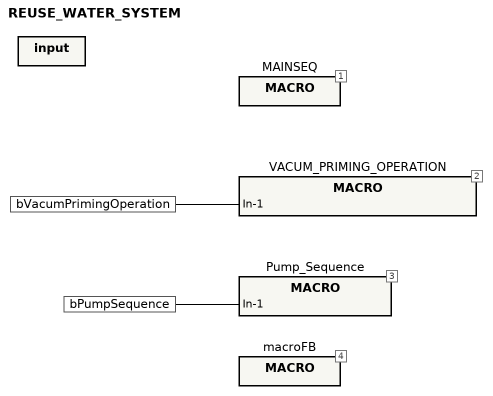
[picture p24: REUSE_WATER_SYSTEM (CFC)]
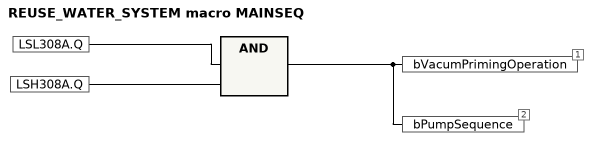
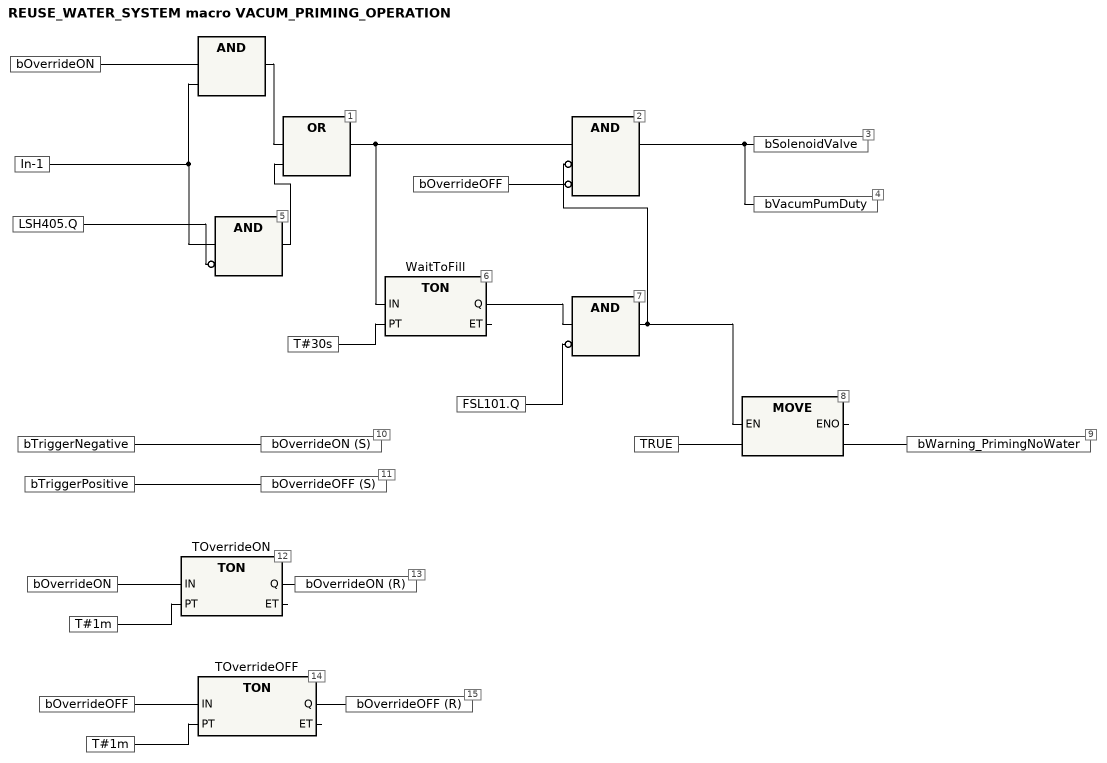
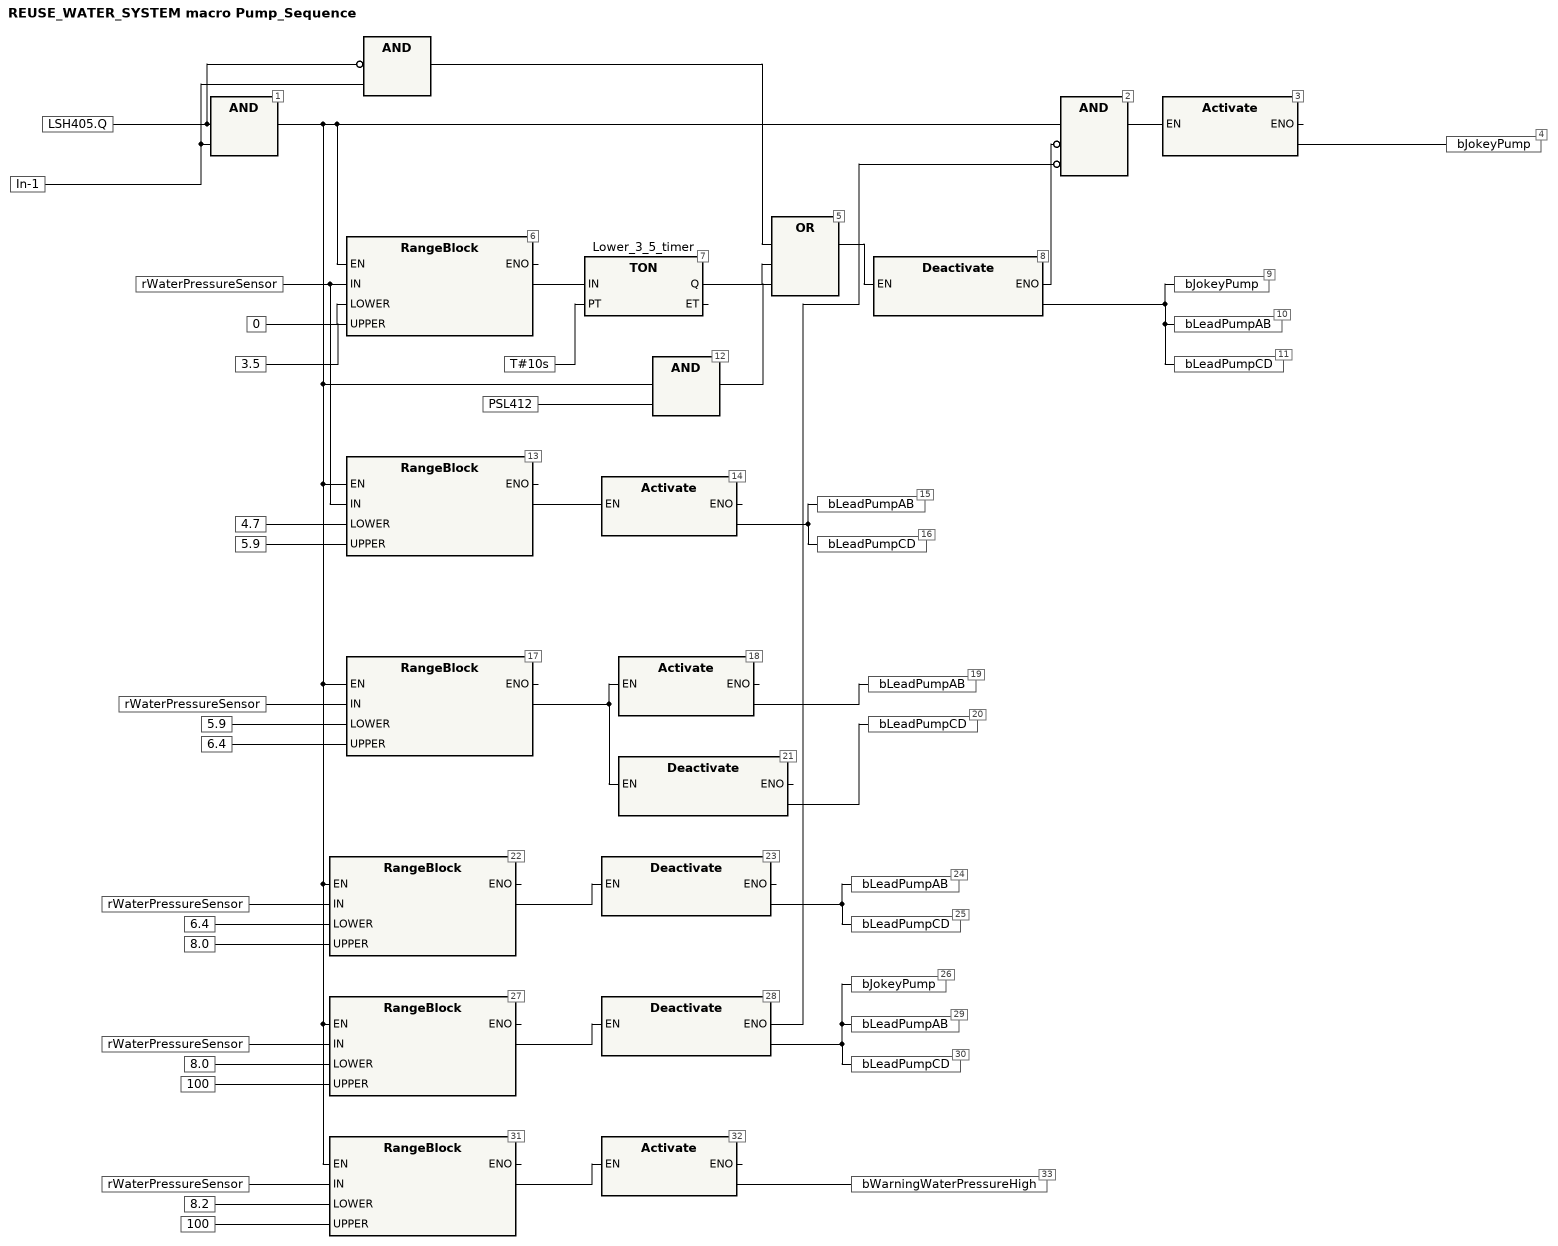
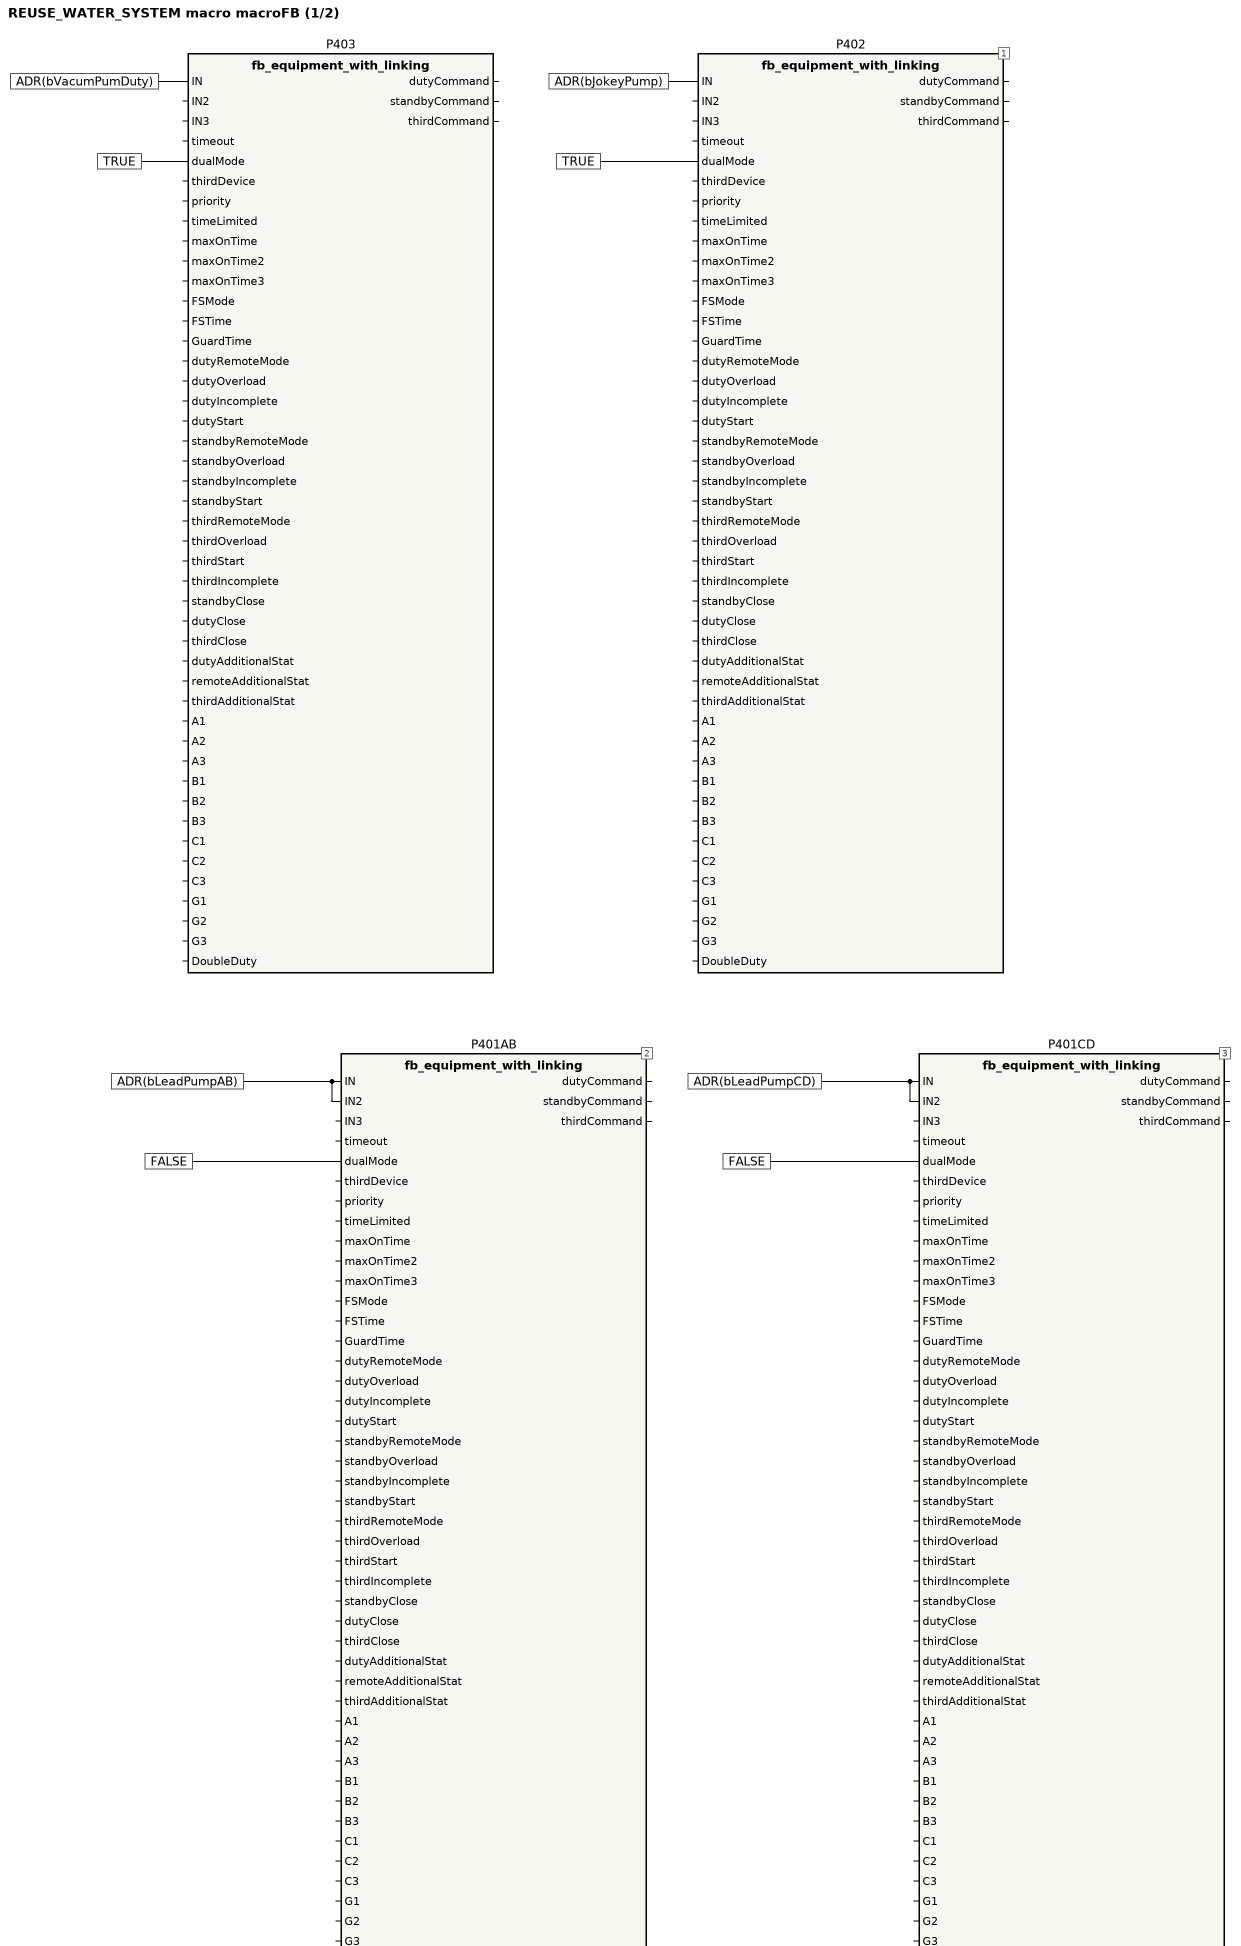
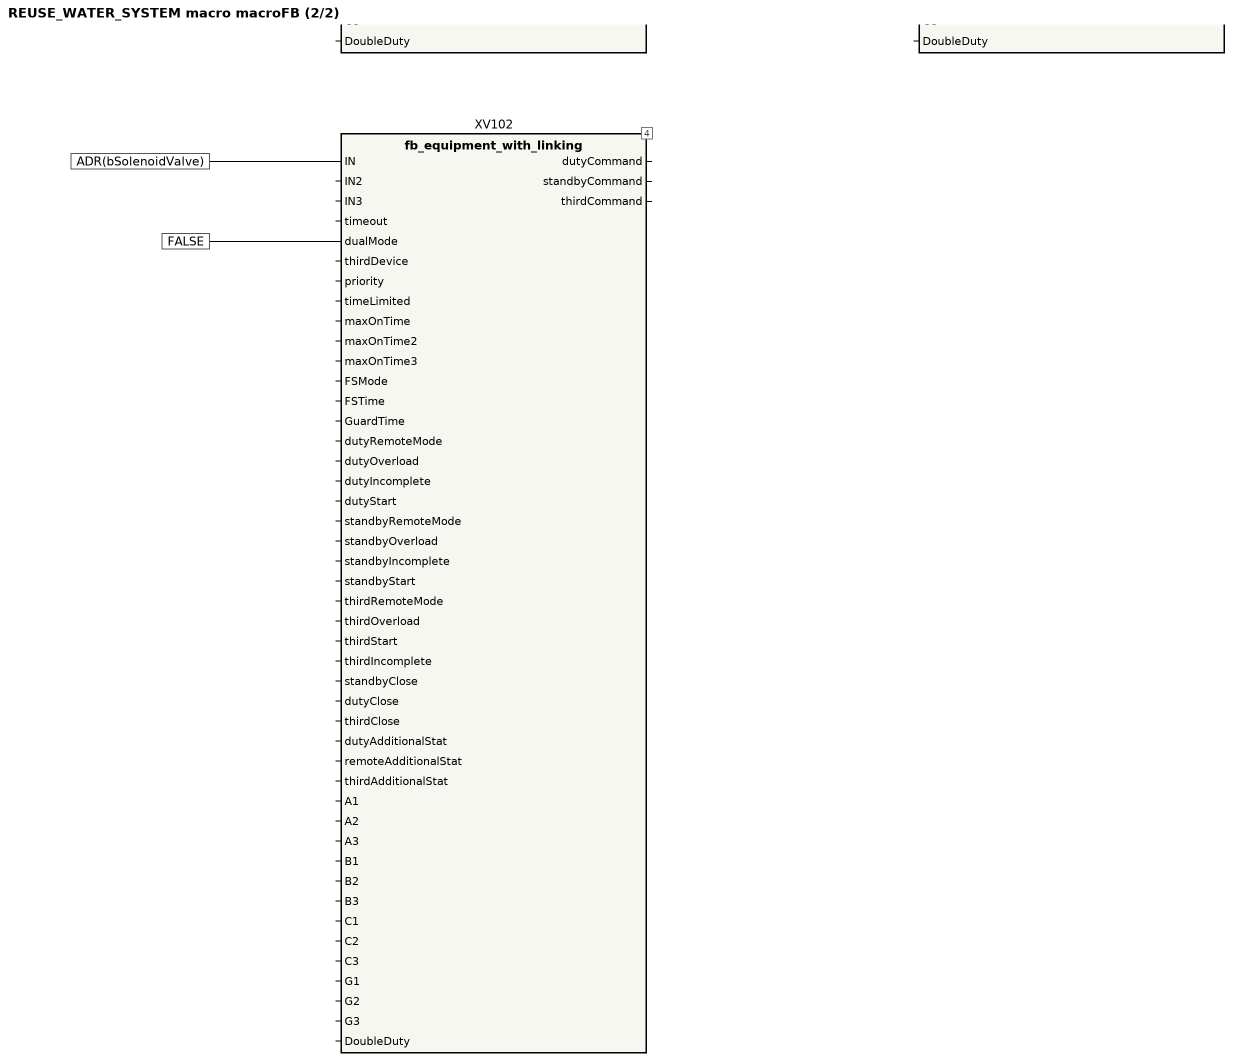
_CFC_ (* Continuous Function Chart, elements in execution order *)
#0 input()
#1 MACRO MAINSEQ()
	#2 AND(LSL308A.Q, LSH308A.Q)
	#3 bVacumPrimingOperation <= #2
	#4 bPumpSequence <= #2
END_MACRO
#5 MACRO VACUM_PRIMING_OPERATION(pin 1 "In-1": bVacumPrimingOperation)
	#6 AND(bOverrideON, pin 1)
	#7 OR(#6, #11)
	#8 AND(#7, NOT #13, NOT bOverrideOFF)
	#9 bSolenoidValve <= #8
	#10 bVacumPumDuty <= #8
	#11 AND(pin 1, NOT LSH405.Q)
	#12 WaitToFill:TON(IN: #7, PT: T#30s)
	#13 AND(#12.Q, NOT FSL101.Q)
	#14 MOVE(EN: #13, TRUE)
	#15 bWarning_PrimingNoWater <= #14
	#16 S bOverrideON <= bTriggerNegative
	#17 S bOverrideOFF <= bTriggerPositive
	#18 TOverrideON:TON(IN: bOverrideON, PT: T#1m)
	#19 R bOverrideON <= #18.Q
	#20 TOverrideOFF:TON(IN: bOverrideOFF, PT: T#1m)
	#21 R bOverrideOFF <= #20.Q
END_MACRO
#22 MACRO Pump_Sequence(pin 1 "In-1": bPumpSequence)
	#23 AND(NOT LSH405.Q, pin 1)
	#24 AND(LSH405.Q, pin 1)
	#25 AND(#24, NOT #31.ENO, NOT #51.ENO)
	#26 Activate(EN: #25)
	#27 bJokeyPump <= #26
	#28 OR(#23, #30.Q, #35)
	#29 RangeBlock(EN: #24, IN: rWaterPressureSensor, LOWER: 0, UPPER: 3.5)
	#30 Lower_3_5_timer:TON(IN: #29, PT: T#10s)
	#31 Deactivate(EN: #28)
	#32 bJokeyPump <= #31
	#33 bLeadPumpAB <= #31
	#34 bLeadPumpCD <= #31
	#35 AND(#24, PSL412)
	#36 RangeBlock(EN: #24, IN: rWaterPressureSensor, LOWER: 4.7, UPPER: 5.9)
	#37 Activate(EN: #36)
	#38 bLeadPumpAB <= #37
	#39 bLeadPumpCD <= #37
	#40 RangeBlock(EN: #24, IN: rWaterPressureSensor, LOWER: 5.9, UPPER: 6.4)
	#41 Activate(EN: #40)
	#42 bLeadPumpAB <= #41
	#43 bLeadPumpCD <= #44
	#44 Deactivate(EN: #40)
	#45 RangeBlock(EN: #24, IN: rWaterPressureSensor, LOWER: 6.4, UPPER: 8.0)
	#46 Deactivate(EN: #45)
	#47 bLeadPumpAB <= #46
	#48 bLeadPumpCD <= #46
	#49 bJokeyPump <= #51
	#50 RangeBlock(EN: #24, IN: rWaterPressureSensor, LOWER: 8.0, UPPER: 100)
	#51 Deactivate(EN: #50)
	#52 bLeadPumpAB <= #51
	#53 bLeadPumpCD <= #51
	#54 RangeBlock(EN: #24, IN: rWaterPressureSensor, LOWER: 8.2, UPPER: 100)
	#55 Activate(EN: #54)
	#56 bWarningWaterPressureHigh <= #55
END_MACRO
#57 MACRO macroFB()
	#58 P403:fb_equipment_with_linking(IN: ADR(bVacumPumDuty), IN2: -, IN3: -, timeout: -, dualMode: TRUE, thirdDevice: -, priority: -, timeLimited: -, maxOnTime: -, maxOnTime2: -, maxOnTime3: -, FSMode: -, FSTime: -, GuardTime: -, dutyRemoteMode: -, dutyOverload: -, dutyIncomplete: -, dutyStart: -, standbyRemoteMode: -, standbyOverload: -, standbyIncomplete: -, standbyStart: -, thirdRemoteMode: -, thirdOverload: -, thirdStart: -, thirdIncomplete: -, standbyClose: -, dutyClose: -, thirdClose: -, dutyAdditionalStat: -, remoteAdditionalStat: -, thirdAdditionalStat: -, A1: -, A2: -, A3: -, B1: -, B2: -, B3: -, C1: -, C2: -, C3: -, G1: -, G2: -, G3: -, DoubleDuty: -)
	#59 P402:fb_equipment_with_linking(IN: ADR(bJokeyPump), IN2: -, IN3: -, timeout: -, dualMode: TRUE, thirdDevice: -, priority: -, timeLimited: -, maxOnTime: -, maxOnTime2: -, maxOnTime3: -, FSMode: -, FSTime: -, GuardTime: -, dutyRemoteMode: -, dutyOverload: -, dutyIncomplete: -, dutyStart: -, standbyRemoteMode: -, standbyOverload: -, standbyIncomplete: -, standbyStart: -, thirdRemoteMode: -, thirdOverload: -, thirdStart: -, thirdIncomplete: -, standbyClose: -, dutyClose: -, thirdClose: -, dutyAdditionalStat: -, remoteAdditionalStat: -, thirdAdditionalStat: -, A1: -, A2: -, A3: -, B1: -, B2: -, B3: -, C1: -, C2: -, C3: -, G1: -, G2: -, G3: -, DoubleDuty: -)
	#60 P401AB:fb_equipment_with_linking(IN: ADR(bLeadPumpAB), IN2: ADR(bLeadPumpAB), IN3: -, timeout: -, dualMode: FALSE, thirdDevice: -, priority: -, timeLimited: -, maxOnTime: -, maxOnTime2: -, maxOnTime3: -, FSMode: -, FSTime: -, GuardTime: -, dutyRemoteMode: -, dutyOverload: -, dutyIncomplete: -, dutyStart: -, standbyRemoteMode: -, standbyOverload: -, standbyIncomplete: -, standbyStart: -, thirdRemoteMode: -, thirdOverload: -, thirdStart: -, thirdIncomplete: -, standbyClose: -, dutyClose: -, thirdClose: -, dutyAdditionalStat: -, remoteAdditionalStat: -, thirdAdditionalStat: -, A1: -, A2: -, A3: -, B1: -, B2: -, B3: -, C1: -, C2: -, C3: -, G1: -, G2: -, G3: -, DoubleDuty: -)
	#61 P401CD:fb_equipment_with_linking(IN: ADR(bLeadPumpCD), IN2: ADR(bLeadPumpCD), IN3: -, timeout: -, dualMode: FALSE, thirdDevice: -, priority: -, timeLimited: -, maxOnTime: -, maxOnTime2: -, maxOnTime3: -, FSMode: -, FSTime: -, GuardTime: -, dutyRemoteMode: -, dutyOverload: -, dutyIncomplete: -, dutyStart: -, standbyRemoteMode: -, standbyOverload: -, standbyIncomplete: -, standbyStart: -, thirdRemoteMode: -, thirdOverload: -, thirdStart: -, thirdIncomplete: -, standbyClose: -, dutyClose: -, thirdClose: -, dutyAdditionalStat: -, remoteAdditionalStat: -, thirdAdditionalStat: -, A1: -, A2: -, A3: -, B1: -, B2: -, B3: -, C1: -, C2: -, C3: -, G1: -, G2: -, G3: -, DoubleDuty: -)
	#62 XV102:fb_equipment_with_linking(IN: ADR(bSolenoidValve), IN2: -, IN3: -, timeout: -, dualMode: FALSE, thirdDevice: -, priority: -, timeLimited: -, maxOnTime: -, maxOnTime2: -, maxOnTime3: -, FSMode: -, FSTime: -, GuardTime: -, dutyRemoteMode: -, dutyOverload: -, dutyIncomplete: -, dutyStart: -, standbyRemoteMode: -, standbyOverload: -, standbyIncomplete: -, standbyStart: -, thirdRemoteMode: -, thirdOverload: -, thirdStart: -, thirdIncomplete: -, standbyClose: -, dutyClose: -, thirdClose: -, dutyAdditionalStat: -, remoteAdditionalStat: -, thirdAdditionalStat: -, A1: -, A2: -, A3: -, B1: -, B2: -, B3: -, C1: -, C2: -, C3: -, G1: -, G2: -, G3: -, DoubleDuty: -)
END_MACRO
_END_CFC_
(* the same logic as Structured Text *)
input();
(* macro MAINSEQ *)
bVacumPrimingOperation := LSL308A.Q AND LSH308A.Q;
bPumpSequence := LSL308A.Q AND LSH308A.Q;
(* macro VACUM_PRIMING_OPERATION *)
_t1 := (bOverrideON AND bVacumPrimingOperation) OR _t23;
_t4 := _t1 AND NOT _t10 AND NOT bOverrideOFF;
bSolenoidValve := _t4;
bVacumPumDuty := _t4;
_t23 := bVacumPrimingOperation AND NOT LSH405.Q;
WaitToFill(IN := _t1, PT := T#30s);
_t10 := WaitToFill.Q AND NOT FSL101.Q;
IF _t10 THEN bWarning_PrimingNoWater := TRUE; END_IF;
IF bTriggerNegative THEN bOverrideON := TRUE; END_IF;
IF bTriggerPositive THEN bOverrideOFF := TRUE; END_IF;
TOverrideON(IN := bOverrideON, PT := T#1m);
IF TOverrideON.Q THEN bOverrideON := FALSE; END_IF;
TOverrideOFF(IN := bOverrideOFF, PT := T#1m);
IF TOverrideOFF.Q THEN bOverrideOFF := FALSE; END_IF;
(* macro Pump_Sequence *)
_t109 := NOT LSH405.Q AND bPumpSequence;
_t44 := LSH405.Q AND bPumpSequence;
IF _t44 AND NOT _en56 AND NOT _en89 THEN bJokeyPump := Activate(); END_IF;
_t101 := _t109 OR Lower_3_5_timer.Q OR _t102;
IF _t44 THEN _t49 := RangeBlock(IN := rWaterPressureSensor, LOWER := 0, UPPER := 3.5); END_IF;
Lower_3_5_timer(IN := _t49, PT := T#10s);
_en56 := _t101;
IF _en56 THEN _t56 := Deactivate(); END_IF;
IF _en56 THEN bJokeyPump := _t56; END_IF;
IF _en56 THEN bLeadPumpAB := _t56; END_IF;
IF _en56 THEN bLeadPumpCD := _t56; END_IF;
_t102 := _t44 AND PSL412;
IF _t44 THEN _t62 := RangeBlock(IN := rWaterPressureSensor, LOWER := 4.7, UPPER := 5.9); END_IF;
_en65 := _t62;
IF _en65 THEN _t65 := Activate(); END_IF;
IF _en65 THEN bLeadPumpAB := _t65; END_IF;
IF _en65 THEN bLeadPumpCD := _t65; END_IF;
IF _t44 THEN _t68 := RangeBlock(IN := rWaterPressureSensor, LOWER := 5.9, UPPER := 6.4); END_IF;
IF _t68 THEN bLeadPumpAB := Activate(); END_IF;
bLeadPumpCD := _t73;
IF _t68 THEN _t73 := Deactivate(); END_IF;
IF _t44 THEN _t77 := RangeBlock(IN := rWaterPressureSensor, LOWER := 6.4, UPPER := 8.0); END_IF;
_en78 := _t77;
IF _en78 THEN _t78 := Deactivate(); END_IF;
IF _en78 THEN bLeadPumpAB := _t78; END_IF;
IF _en78 THEN bLeadPumpCD := _t78; END_IF;
bJokeyPump := _t89;
IF _t44 THEN _t88 := RangeBlock(IN := rWaterPressureSensor, LOWER := 8.0, UPPER := 100); END_IF;
_en89 := _t88;
IF _en89 THEN _t89 := Deactivate(); END_IF;
bLeadPumpAB := _t89;
bLeadPumpCD := _t89;
IF _t44 THEN _t97 := RangeBlock(IN := rWaterPressureSensor, LOWER := 8.2, UPPER := 100); END_IF;
IF _t97 THEN bWarningWaterPressureHigh := Activate(); END_IF;
(* macro macroFB *)
P403(IN := ADR(bVacumPumDuty), dualMode := TRUE);
P402(IN := ADR(bJokeyPump), dualMode := TRUE);
P401AB(IN := ADR(bLeadPumpAB), IN2 := ADR(bLeadPumpAB), dualMode := FALSE);
P401CD(IN := ADR(bLeadPumpCD), IN2 := ADR(bLeadPumpCD), dualMode := FALSE);
XV102(IN := ADR(bSolenoidValve), dualMode := FALSE);
END_PROGRAM
ACTION input:
LSH405();
LSL308A();
LSH308A();

rWaterPressureSensor := INT_TO_REAL(PSL411)*(10.0/32767.0);
END_ACTION

(* POU module/Deactivate, ST *)
FUNCTION Deactivate : BOOL
VAR_INPUT
END_VAR
VAR
END_VAR
Deactivate := FALSE;
END_FUNCTION

(* POU SLUDGE_TANK, CFC *)
PROGRAM SLUDGE_TANK
VAR
END_VAR
_CFC_ (* Continuous Function Chart, elements in execution order *)
_END_CFC_
END_PROGRAM

(* POU module/TANK_FOR_STREAM_1, ST *)
PROGRAM TANK_FOR_STREAM_1
VAR

(* ---------------------------------------- INLET EQ PUMP OPERATION------------------------------------*)
	LSD101A : inBlock;
	LSL101A : inBlock;
	LSS101A : inBlock;
	LSH101A : inBlock;
	LSHH105A : inBlock;
	LSH103A : inBlock;

	P101A: BOOL;

	warning_EQFloatSensorDry: BOOL;
	critical_EQFloatSensorDry: BOOL;
	critical_EQFloatSensorHi: BOOL;

	fbP101A : fb_equipment;
	P101A1RemoteMode AT%I*: BOOL;
	P101A1Overload AT%I*: BOOL;
	P101A1Incomplete AT%I*: BOOL;
	P101A1Started AT%I*: BOOL;
	P101A2RemoteMode AT%I*: BOOL;
	P101A2Overload AT%I*: BOOL;
	P101A2Incomplete AT%I*: BOOL;
	P101A2Started AT%I*: BOOL;
	warning_P101A1Overload: BOOL;
	warning_P101A1Failed: BOOL;
	warning_P101A2Overload: BOOL;
	warning_P101A2Failed: BOOL;
	critical_P101AStartingFailed: BOOL;
	critical_P101A1StopFailed: BOOL;
	critical_P101A2StopFailed: BOOL;

	P101A1Command AT%Q*: BOOL;
	P101A2Command AT%Q*: BOOL;


(*--------------------------------------------------MIXER Operation-------------------------------------------------*)
	fbM101A : fb_equipment;
	M101A : BOOL;

	M101A1RemoteMode AT%I*: BOOL;
	M101A1Overload AT%I*: BOOL;
	M101A1Incomplete AT%I*: BOOL;
	M101A1Started AT%I*: BOOL;
	M101A2RemoteMode AT%I*: BOOL;
	M101A2Overload AT%I*: BOOL;
	M101A2Incomplete AT%I*: BOOL;
	M101A2Started AT%I*: BOOL;
	warning_M101A1Overload: BOOL;
	warning_M101A1Failed: BOOL;
	warning_M101A2Overload: BOOL;
	warning_M101A2Failed: BOOL;
	critical_M101AStartingFailed: BOOL;
	critical_M101A1StopFailed: BOOL;
	critical_M101A2StopFailed: BOOL;

	M101A1Command AT%Q*: BOOL;
	M101A2Command AT%Q*: BOOL;

	LSL100A : inBlock;
	LSHL100A : inBlock;



END_VAR
LSD101A();
LSL101A();
LSS101A();
LSH101A();
LSHH105A();
LSH103A();

LSL100A();
LSHL100A();



(* ---------------------------------------- INLET EQ PUMP OPERATION------------------------------------*)
fbP101A.IN := ADR(P101A);


IF LSL101A.Q THEN
	IF LSS101A.Q THEN
		P101A:=TRUE;
		IF LSH101A.Q THEN
			critical_EQFloatSensorHi := TRUE;
			IF LSHH105A.Q OR LSH103A.Q THEN
				P101A:=FALSE;
			END_IF
		END_IF
	ELSE
		P101A:=FALSE;
	END_IF
ELSE
	P101A:=FALSE;
	IF LSD101A.Q	THEN
		warning_EQFloatSensorDry :=TRUE;
	ELSE
		critical_EQFloatSensorDry := TRUE;
	END_IF
END_IF

fbP101A(
	dutyRemoteMode:= P101A1RemoteMode,
	dutyOverload:=P101A1Overload ,
	dutyIncomplete:=P101A1Incomplete ,
	dutyStart:=P101A1Started ,
	standbyRemoteMode:=P101A2RemoteMode ,
	standbyOverload:=P101A2Overload ,
	standbyIncomplete:=P101A2Incomplete  ,
	standbyStart:=P101A2Started ,
	timeout:=T#2s ,
	dualMode:= TRUE,
	warningDutyOverload:=ADR(warning_P101A1Overload) ,
	warningDutyFailed:=ADR(warning_P101A1Failed) ,
	warningStandbyOverload:=ADR(warning_P101A2Overload) ,
	warningStandbyFailed:=ADR(warning_P101A2Failed) ,
	criticalErrorStartingFailed:=ADR(critical_P101AStartingFailed) ,
	criticalDutyStopFailed:= ADR(critical_P101A1StopFailed),
	criticalStandbyStopFailed:=ADR(critical_P101A2StopFailed),
	dutyCommand=>P101A1Command ,
	standbyCommand=>P101A2Command);

(*--------------------------------------------------MIXER Operation-------------------------------------------------*)
fbM101A.IN:=ADR(M101A);

IF LSL100A.Q THEN
	IF LSHL100A.Q THEN
		M101A:=TRUE ;
	ELSE
		M101A:=FALSE;
	END_IF
ELSE
	M101A:=FALSE;
END_IF


fbM101A(
	dutyRemoteMode:= M101A1RemoteMode,
	dutyOverload:=M101A1Overload ,
	dutyIncomplete:=M101A1Incomplete ,
	dutyStart:=M101A1Started ,
	standbyRemoteMode:=M101A2RemoteMode ,
	standbyOverload:=M101A2Overload ,
	standbyIncomplete:=M101A2Incomplete  ,
	standbyStart:=M101A2Started ,
	timeout:=T#2s ,
	dualMode:= TRUE,
	warningDutyOverload:=ADR(warning_M101A1Overload) ,
	warningDutyFailed:=ADR(warning_M101A1Failed) ,
	warningStandbyOverload:=ADR(warning_M101A2Overload) ,
	warningStandbyFailed:=ADR(warning_M101A2Failed) ,
	criticalErrorStartingFailed:=ADR(critical_M101AStartingFailed) ,
	criticalDutyStopFailed:= ADR(critical_M101A1StopFailed),
	criticalStandbyStopFailed:=ADR(critical_M101A2StopFailed),
	dutyCommand=>M101A1Command ,
	standbyCommand=>M101A2Command );
END_PROGRAM

(* POU module/fb_equipment, ST *)
FUNCTION_BLOCK fb_equipment
VAR_INPUT
	IN							: POINTER TO BOOL;
	dutyRemoteMode				: BOOL;
	dutyOverload					: BOOL;
	dutyIncomplete				: BOOL;
	dutyStart						: BOOL;

	standbyRemoteMode			: BOOL;
	standbyOverload				: BOOL;
	standbyIncomplete			: BOOL;
	standbyStart					: BOOL;

	thirdRemoteMode				: BOOL;
	thirdOverload					: BOOL;
	thirdStart						: BOOL;
	thirdIncomplete				: BOOL;

	standbyClose					: BOOL;
	dutyClose					: BOOL;
	thirdClose					: BOOL;

	dutyAdditionalStat				: BOOL := TRUE;
	remoteAdditionalStat			: BOOL := TRUE;
	thirdAdditionalStat				: BOOL := TRUE;

	timeout						: TIME:= T#2s;
	dualMode					: BOOL:=TRUE;
	thirdDevice					: BOOL:= FALSE;
	priority						: BOOL := FALSE;
	timeLimited					: BOOL :=FALSE;
	maxOnTime					: TIME := T#10s;
	maxOnTime2					: TIME := T#10s;
	maxOnTime3					: TIME := T#10s;

	FSMode						: BOOL := FALSE;
	FSTime						: TIME := T#2m;
(*
	FSBothTime					: TIME := T#5m;
*)
	GuardTime					: TIME := T#5m;

	A1							: POINTER TO BOOL;
	A2							: POINTER TO BOOL;
	A3							: POINTER TO BOOL;
	B1							: POINTER TO BOOL;
	B2							: POINTER TO BOOL;
	B3							: POINTER TO BOOL;
	C1							: POINTER TO BOOL;
	C2							: POINTER TO BOOL;
	C3							: POINTER TO BOOL;
(*
	Q1							: POINTER TO BOOL;
	Q2							: POINTER TO BOOL;
	Q3							: POINTER TO BOOL;
*)
	G1							: POINTER TO BOOL;
	G2							: POINTER TO BOOL;
	G3							: POINTER TO BOOL;

	warningDutyOverload			: POINTER TO BOOL;
	warningDutyFailed				: POINTER TO BOOL;
	warningDutyNotClose			: POINTER TO BOOL;
	warningDutyClose				: POINTER TO BOOL;
	warningStandbyOverload		: POINTER TO BOOL;
	warningStandbyFailed			: POINTER TO BOOL;
	warningStandbyNotClose		: POINTER TO BOOL;
	warningStandbyClose			: POINTER TO BOOL;
	warningThirdOverload			: POINTER TO BOOL;
	warningThirdFailed			: POINTER TO BOOL;
	warningThirdNotClose			: POINTER TO BOOL;
	warningThirdClose			: POINTER TO BOOL;

	criticalErrorStartingFailed		: POINTER TO BOOL;
	criticalDutyStopFailed			: POINTER TO BOOL;
	criticalStandbyStopFailed		: POINTER TO BOOL;
	criticalThirdStopFailed			: POINTER TO BOOL;

END_VAR
VAR_OUTPUT
	dutyCommand				: BOOL;
	standbyCommand				: BOOL;
	thirdCommand				: BOOL;
END_VAR
VAR
	duty							: INT;
	iStopDuty					: INT;
	state						: INT;
	third							: INT;
	iStopThird					: INT;
	iStopStandby					: INT;
	standby						: INT;
	startDuty						: BOOL;
	startStandby					: BOOL;
	stopStandby					: BOOL;
	stopDuty						: BOOL;
	dutyHalt						: BOOL;
	standbyHalt					: BOOL;
	stopThird					: BOOL;
	startThird					: BOOL;
	thirdHalt						: BOOL;

	dutyTimer					: TON;
	standbyTimer					: TON;
	stopStandbyTimer				: TON;
	stopDutyTimer				: TON;
	FSStopDuty					:TON;
	FSStopStandby				: TON;
	FSBothStop					: TON;
	OnTimer						: TON;
	StandbyOnTimer				: TON;
	thirdTimer					: TON;
	stopThirdTimer				: TON;
	GuardTONDuty				: TON;
	GuardTONStandby			: TON;
	GuardTONThird				: TON;

	ROnce5						: R_TRIG;
	ROnce10					: R_TRIG;
	ROnce20					: R_TRIG;
	SOnceDuty					: R_TRIG;
	SOnceStandby				: R_TRIG;
	SOnceFS					: R_TRIG;
	SOnceThird					: R_TRIG;
	DutyStopR					: R_TRIG;
	StandbyStopR				: R_TRIG;
	ThirdStopR					: R_TRIG;

	internalDummy: BOOL;
	dummyIN: BOOL;
END_VAR
VAR_IN_OUT
END_VAR
IF IN = 0 THEN
	IN := ADR(dummyIN);
END_IF

IF A1 = 0 THEN
	A1 := ADR(internalDummy);
END_IF
IF A2 = 0 THEN
	A2 := ADR(internalDummy);
END_IF
IF A3 = 0 THEN
	A3 := ADR(internalDummy);
END_IF

IF B1 = 0 THEN
	B1 := ADR(internalDummy);
END_IF
IF B2 = 0 THEN
	B2 := ADR(internalDummy);
END_IF
IF B3 = 0 THEN
	B3 := ADR(internalDummy);
END_IF

IF C1 = 0 THEN
	C1 := ADR(internalDummy);
END_IF
IF C2 = 0 THEN
	C2 := ADR(internalDummy);
END_IF
IF C3 = 0 THEN
	C3 := ADR(internalDummy);
END_IF

IF G1 = 0 THEN
	G1 := ADR(internalDummy);
END_IF
IF G2 = 0 THEN
	G2 := ADR(internalDummy);
END_IF
IF G3 = 0 THEN
	G3 := ADR(internalDummy);
END_IF



IF warningDutyOverload = 0 THEN
	warningDutyOverload := ADR(internalDummy);
END_IF
IF warningDutyFailed = 0 THEN
	warningDutyFailed := ADR(internalDummy);
END_IF
IF warningDutyNotClose = 0 THEN
	warningDutyNotClose := ADR(internalDummy);
END_IF
IF warningDutyClose = 0 THEN
	warningDutyClose := ADR(internalDummy);
END_IF



IF warningStandbyOverload = 0 THEN
	warningStandbyOverload := ADR(internalDummy);
END_IF
IF warningStandbyFailed = 0 THEN
	warningStandbyFailed := ADR(internalDummy);
END_IF
IF warningStandbyNotClose = 0 THEN
	warningStandbyNotClose := ADR(internalDummy);
END_IF
IF warningStandbyClose = 0 THEN
	warningStandbyClose := ADR(internalDummy);
END_IF


IF warningThirdOverload = 0 THEN
	warningThirdOverload := ADR(internalDummy);
END_IF
IF warningThirdFailed = 0 THEN
	warningThirdFailed := ADR(internalDummy);
END_IF
IF warningThirdNotClose = 0 THEN
	warningThirdNotClose := ADR(internalDummy);
END_IF
IF warningThirdClose = 0 THEN
	warningThirdClose := ADR(internalDummy);
END_IF


IF criticalErrorStartingFailed = 0 THEN
	criticalErrorStartingFailed := ADR(internalDummy);
END_IF
IF criticalDutyStopFailed = 0 THEN
	criticalDutyStopFailed := ADR(internalDummy);
END_IF
IF criticalStandbyStopFailed = 0 THEN
	criticalStandbyStopFailed := ADR(internalDummy);
END_IF
IF criticalThirdStopFailed = 0 THEN
	criticalThirdStopFailed := ADR(internalDummy);
END_IF

(*---------------------------------------------------------------------------------------------------------------------------*)

IF NOT IN^ THEN
	state := 0;
	stopDuty := TRUE;
	stopStandby := TRUE;

	startDuty:=FALSE;
	startStandby := FALSE;
	IF thirdDevice THEN
		stopThird :=TRUE;
		startThird := FALSE;
	END_IF
ELSIF IN^ AND NOT dualMode THEN
	state := 0;
	stopDuty := FALSE;
	stopStandby := FALSE;

	startDuty:=TRUE;
	startStandby := TRUE;
	IF thirdDevice THEN
		stopThird :=FALSE;
		startThird := TRUE;
	END_IF

	A1^:= TRUE;
	A2^:=TRUE;
	A3^ :=TRUE;
	B1^:= TRUE;
	B2^:=TRUE;
	B3^ :=TRUE;
	C1^:= TRUE;
	C2^:=TRUE;
	C3^ :=TRUE;
END_IF

(*-------------------------------------------------------------------------------------------------------------------------------------------*)

CASE state OF
0:
	state := 5;
5:
	IF NOT DutyHalt AND dutyStart THEN
		stopStandby := TRUE;
		stopThird:=TRUE;
	END_IF

	stopDuty := FALSE;
	startDuty := TRUE;
	IF timeLimited THEN
		OnTimer(IN:=TRUE,PT:=maxOnTime);
	ELSE
		OnTimer(IN:=FALSE,PT:=maxOnTime);
	END_IF
	IF dutyHalt  OR onTimer.Q THEN
		OnTimer(IN:=FALSE,PT:=maxOnTime);
		startDuty := FALSE;
		stopDuty := TRUE;
		state := 10;
	END_IF
10:
	IF NOT StandbyHalt AND standbyStart THEN
		stopDuty := TRUE;
		stopThird:=TRUE;
	END_IF

	stopStandby := FALSE;
	startStandby := TRUE;

	IF timeLimited THEN
		OnTimer(IN:=TRUE,PT:=maxOnTime2);
	ELSE
		OnTimer(IN:=FALSE,PT:=maxOnTime2);
	END_IF
	IF standbyHalt OR onTimer.Q THEN
		OnTimer(IN:=FALSE,PT:=maxOnTime2);
		startStandby := FALSE;
		stopStandby := TRUE;
		IF thirdDevice THEN
			IF priority THEN
				IF dutyIncomplete OR dutyOverload THEN
					state:= 20;
				ELSE
					dutyHalt := FALSE;
					standbyHalt := FALSE;
					state:=0;
				END_IF
			ELSE
				state:= 20;
			END_IF
		ELSE
			IF dutyIncomplete OR dutyOverload THEN
				CriticalErrorStartingFailed^ := TRUE;
			END_IF
			state:=0;
			dutyHalt := FALSE;
			standbyHalt := FALSE;
		END_IF
	END_IF
20:
	IF NOT thirdHalt AND thirdStart THEN
		stopStandby := TRUE;
		stopDuty:=TRUE;
	END_IF

	stopThird := FALSE;
	startThird := TRUE;
	IF timeLimited THEN
		OnTimer(IN:=TRUE,PT:=maxOnTime3);
	ELSE
		OnTimer(IN:=FALSE,PT:=maxOnTime3);
	END_IF
	IF thirdHalt OR OnTimer.Q THEN
		OnTimer(IN:=FALSE,PT:=maxOnTime3);
		startThird := FALSE;
		stopThird := TRUE;
		state := 0;
		IF  (dutyIncomplete OR dutyOverload)  AND (standbyIncomplete OR standbyOverload) THEN
				CriticalErrorStartingFailed^ := TRUE;
		END_IF
		dutyHalt := FALSE;
		standbyHalt := FALSE;
		thirdHalt := FALSE;
	END_IF
END_CASE



(*-------------------------------------------------------------------------------------------------------------------------------------------*)

CASE duty OF
0:
	IF startDuty THEN
		duty := 5;
	END_IF
5:
	IF dutyRemoteMode AND dutyAdditionalStat THEN
		duty := 10;
	ELSE
		duty := 900;
	END_IF
10:
	IF dutyOverload THEN
		warningDutyOverload^ := TRUE;
		dutyHalt := TRUE;
		duty := 40;
	ELSE
		duty := 15;
	END_IF

15:
	duty := 20;
	dutyCommand := TRUE;
20:
	dutyTimer(IN:= TRUE, PT := timeout);
	IF dutyTimer.Q THEN
		dutyTimer(IN:=FALSE);
		duty := 30;
	END_IF
30:

		IF dutyIncomplete OR NOT dutyStart THEN
			warningDutyFailed^ := TRUE;
			dutyHalt := TRUE;
			IF  dutyClose THEN
				warningDutyClose^ := TRUE;
			END_IF
		END_IF
		duty := 40;
40:

	duty := 900;
900:
	duty := 0;
END_CASE

(*----------------------------------------------------------------------------------------------------------------------*)

CASE standby OF
0:
	IF startStandby THEN
		standby := 5;
	END_IF
5:
	IF standbyRemoteMode AND remoteAdditionalStat THEN
		standby := 10;
	ELSE
		standby := 900;
	END_IF
10:
	IF standbyOverload THEN
		warningStandbyOverload^ := TRUE;
		standbyHalt := TRUE;
		standby := 40;
	ELSE
		standby := 15;
	END_IF
15:
		standbyCommand := TRUE;
		standby := 20;
20:
	standbyTimer(IN:= TRUE, PT := timeout);
	IF standbyTimer.Q THEN
		standbyTimer(IN:=FALSE);
		standby := 30;
	END_IF
30:

		IF standbyIncomplete OR NOT standbyStart THEN
			warningStandbyFailed^ := TRUE;
			standbyHalt := TRUE;
			IF  standbyClose THEN
				warningStandbyClose^ := TRUE;
			END_IF
		END_IF
		standby := 40;
40:

	standby := 900;

900:
	standby := 0;
END_CASE

(*-------------------------------------------------------------------------------------------------------------------------------------------*)

CASE third OF
0:
	IF startThird THEN
		third := 5;
	END_IF
5:
	IF thirdRemoteMode AND thirdAdditionalStat THEN
		third := 10;
	ELSE
		third := 900;
	END_IF
10:
	IF thirdOverload THEN
		warningThirdOverload^ := TRUE;
		thirdHalt := TRUE;
		third := 40;
	ELSE
		third := 15;
	END_IF
15:
		thirdCommand := TRUE;
		third := 20;
20:
	thirdTimer(IN:= TRUE, PT := timeout);
	IF thirdTimer.Q THEN
		thirdTimer(IN:=FALSE);
		third := 30;
	END_IF
30:

		IF thirdIncomplete OR NOT thirdStart THEN
			warningThirdFailed^ := TRUE;
			thirdHalt := TRUE;
			IF thirdClose THEN
				warningThirdClose^ := TRUE;
			END_IF
		END_IF
		third := 40;
40:

	third := 900;

900:
	third := 0;
END_CASE

(*-------------------------------------------------------------------------------------------------------------------------------------------*)

ROnce5(CLK:=(state=5));
IF ROnce5.Q THEN
		A1^:= TRUE;
		A2^:=TRUE;
		A3^ :=TRUE;
END_IF

ROnce10(CLK:=(state=10));
IF ROnce10.Q THEN
		B1^:= TRUE;
		B2^:= TRUE;
		B3^:= TRUE;
END_IF

IF thirdDevice THEN
ROnce20(CLK:=(state=20));
IF ROnce20.Q THEN
		C1^:= TRUE;
		C2^:= TRUE;
		C3^:= TRUE;
END_IF
END_IF

(*-------------------------------------------------------------------------------------------------------------------------------------------*)
GuardTONDuty(IN:=dutyIncomplete OR dutyOverload OR NOT dutyStart, PT:= GuardTime);
IF GuardTONDuty.Q THEN
	G1^ := TRUE;
END_IF
GuardTONStandby(IN:=standbyIncomplete OR standbyOverload OR NOT standbyStart, PT:= GuardTime);
IF GuardTONStandby.Q THEN
	G2^ := TRUE;
END_IF

IF thirdDevice THEN
GuardTONThird(IN:=thirdIncomplete OR thirdOverload OR NOT thirdStart, PT:= GuardTime);
IF GuardTONThird.q THEN
	G3^ := TRUE;
END_IF
END_IF
(*-------------------------------------------------------------------------------------------------------------------------------------------*)
stopAction;
test();
END_FUNCTION_BLOCK
ACTION stopAction:
CASE iStopDuty OF
0:
(*
	DutyStopR(CLK:=stopDuty);
	IF DutyStopR.Q THEN
		iStopDuty := 5;
	END_IF


5:
*)
	IF FSMode THEN
		FSStopDuty(IN:=TRUE,PT:=FSTime);
		IF FSStopDuty.Q THEN
			iStopDuty := 10;
			FSStopDuty(IN:=FALSE,PT:=FSTime);
		END_IF
	ELSE
		iStopDuty:=10;
	END_IF
10:
	dutyCommand := FALSE;
	stopDutyTimer(IN:=TRUE, PT:=timeout);
		IF stopDutyTimer.Q THEN
			stopDutyTimer(IN:=FALSE);
			IF NOT dutyClose THEN
				IF dutyStart THEN
					criticalDutyStopFailed^ := TRUE;
				END_IF
				warningDutyNotClose^ := TRUE;
			END_IF
			iStopDuty := 0;
		END_IF
END_CASE

(*-------------------------------------------------------------------------------------------------------------------------------------------*)

CASE iStopStandby OF
0:
(*
	StandbyStopR(CLK:=stopStandby);
	IF StandbyStopR.Q THEN
		iStopStandby := 5;
	END_IF
5:
*)
	IF FSMode THEN
		FSStopStandby(IN:=TRUE,PT:=FSTime);
		IF FSStopStandby.Q THEN
			iStopStandby := 10;
			FSStopStandby(IN:=FALSE,PT:=FSTime);
		END_IF
	ELSE
		iStopStandby:=10;
	END_IF
10:
	standbyCommand := FALSE;
	stopStandbyTimer(IN:=TRUE, PT:=timeout);
		IF stopStandbyTimer.Q THEN
			stopStandbyTimer(IN:=FALSE);
			IF NOT standbyClose THEN
				IF standbyStart THEN
					criticalStandbyStopFailed^ := TRUE;
				END_IF
					warningStandbyNotClose^ := TRUE;
			END_IF
			iStopStandby := 0;
		END_IF
END_CASE


(*-------------------------------------------------------------------------------------------------------------------------------------------*)

CASE iStopThird OF
0:
(*
	ThirdStopR(CLK:=stopThird);
	IF ThirdStopR.Q THEN
		iStopThird := 10;
	END_IF
10:
*)
	thirdCommand := FALSE;
	stopThirdTimer(IN:=TRUE, PT:=timeout);
		IF stopThirdTimer.Q THEN
			stopThirdTimer(IN:=FALSE);
			IF NOT thirdClose THEN
				IF thirdStart THEN
					criticalThirdStopFailed^ := TRUE;
				END_IF
				warningThirdNotClose^ := TRUE;
			END_IF
			iStopThird := 0;
		END_IF
END_CASE


(*-------------------------------------------------------------------------------------------------------------------------------------------*)

SOnceDuty(CLK:=(iStopDuty = 10));
IF SOnceDuty.Q THEN
		A1^:=FALSE;
		A2^:=FALSE;
		A3^:=FALSE;
END_IF


SOnceStandby(CLK:=(iStopStandby = 10));
IF SOnceStandby.Q THEN
		B1^:=FALSE;
		B2^:=FALSE;
		B3^:=FALSE;
END_IF

IF thirdDevice THEN
SOnceThird(CLK:=(iStopThird = 10));
IF SOnceThird.Q THEN
		C1^:= FALSE;
		C1^:=FALSE;
		C2^:=FALSE;
		C3^:=FALSE;
END_IF
END_IF


(*-------------------------------------------------------------------------------------------------------------------------------------------*)

(*
IF FSMode THEN

FSBothStop(IN:=NOT dutyCommand AND NOT standbyCommand,PT:=FSBothTime);
SOnceFS(CLK:=FSBothStop.Q);
IF SOnceFS.Q THEN
	FSBothStop(IN:=FALSE,PT:=FSBothTime);
	Q1^ := TRUE;
	Q2^ := TRUE;
	Q3^:=TRUE;
END_IF

END_IF
*)
END_ACTION
ACTION test:
dutyStart := dutyCommand;
standbyStart := standbyCommand;
thirdStart:=thirdCommand;
END_ACTION

(* POU module/TANK_FOR_STREAM_2, ST *)
PROGRAM TANK_FOR_STREAM_2
VAR

(* ---------------------------------------- INLET EQ PUMP OPERATION------------------------------------*)
	LSD101B : inBlock;
	LSL101B : inBlock;
	LSS101B : inBlock;
	LSH101B : inBlock;
	LSHH105B : inBlock;
	LSH103B : inBlock;

	P101B: BOOL;

	warning_EQFloatSensorDry: BOOL;
	critical_EQFloatSensorDry: BOOL;
	critical_EQFloatSensorHi: BOOL;

	fbP101B : fb_equipment;
	P101B1RemoteMode AT%I*: BOOL;
	P101B1Overload AT%I*: BOOL;
	P101B1Incomplete AT%I*: BOOL;
	P101B1Started AT%I*: BOOL;
	P101B2RemoteMode AT%I*: BOOL;
	P101B2Overload AT%I*: BOOL;
	P101B2Incomplete AT%I*: BOOL;
	P101B2Started AT%I*: BOOL;
	warning_P101B1Overload: BOOL;
	warning_P101B1Failed: BOOL;
	warning_P101B2Overload: BOOL;
	warning_P101B2Failed: BOOL;
	critical_P101BStartingFailed: BOOL;
	critical_P101B1StopFailed: BOOL;
	critical_P101B2StopFailed: BOOL;

	P101B1Command AT%Q*: BOOL;
	P101B2Command AT%Q*: BOOL;


(*--------------------------------------------------MIXER Operation-------------------------------------------------*)
	fbM101B : fb_equipment;
	M101B : BOOL;

	M101B1RemoteMode AT%I*: BOOL;
	M101B1Overload AT%I*: BOOL;
	M101B1Incomplete AT%I*: BOOL;
	M101B1Started AT%I*: BOOL;
	M101B2RemoteMode AT%I*: BOOL;
	M101B2Overload AT%I*: BOOL;
	M101B2Incomplete AT%I*: BOOL;
	M101B2Started AT%I*: BOOL;

	warning_M101B1Overload: BOOL;
	warning_M101B1Failed: BOOL;
	warning_M101B2Overload: BOOL;
	warning_M101B2Failed: BOOL;
	critical_M101BStartingFailed: BOOL;
	critical_M101B1StopFailed: BOOL;
	critical_M101B2StopFailed: BOOL;

	M101B1Command AT%Q*: BOOL;
	M101B2Command AT%Q*: BOOL;

	LSL100B : inBlock;
	LSHL100B : inBlock;


END_VAR
LSD101B();
LSL101B();
LSS101B();
LSH101B();
LSHH105B();
LSH103B();

LSL100B();
LSHL100B();



(* ---------------------------------------- INLET EQ PUMP OPERATION------------------------------------*)
fbP101B.IN := ADR(P101B);


IF LSL101B.Q THEN
	IF LSS101B.Q THEN
		P101B:=TRUE;
		IF LSH101B.Q THEN
			critical_EQFloatSensorHi := TRUE;
			IF LSHH105B.Q OR LSH103B.Q THEN
				P101B:=FALSE;
			END_IF
		END_IF
	ELSE
		P101B:=FALSE;
	END_IF
ELSE
	P101B:=FALSE;
	IF LSD101B.Q	THEN
		warning_EQFloatSensorDry :=TRUE;
	ELSE
		critical_EQFloatSensorDry := TRUE;
	END_IF
END_IF

fbP101B(
	dutyRemoteMode:= P101B1RemoteMode,
	dutyOverload:=P101B1Overload ,
	dutyIncomplete:=P101B1Incomplete ,
	dutyStart:=P101B1Started ,
	standbyRemoteMode:=P101B2RemoteMode ,
	standbyOverload:=P101B2Overload ,
	standbyIncomplete:=P101B2Incomplete  ,
	standbyStart:=P101B2Started ,
	timeout:=T#2s ,
	dualMode:= TRUE,
	warningDutyOverload:=ADR(warning_P101B1Overload) ,
	warningDutyFailed:=ADR(warning_P101B1Failed) ,
	warningStandbyOverload:=ADR(warning_P101B2Overload) ,
	warningStandbyFailed:=ADR(warning_P101B2Failed) ,
	criticalErrorStartingFailed:=ADR(critical_P101BStartingFailed) ,
	criticalDutyStopFailed:= ADR(critical_P101B1StopFailed),
	criticalStandbyStopFailed:=ADR(critical_P101B2StopFailed),
	dutyCommand=>P101B1Command ,
	standbyCommand=>P101B2Command );

(*--------------------------------------------------MIXER Operation-------------------------------------------------*)
fbM101B.IN := ADR(M101B);

IF LSL100B.Q THEN
	IF LSHL100B.Q THEN
		M101B:=TRUE;
	ELSE
		M101B:=FALSE;
	END_IF
ELSE
	M101B:=FALSE;
END_IF


fbM101B(
	dutyRemoteMode:= M101B1RemoteMode,
	dutyOverload:=M101B1Overload ,
	dutyIncomplete:=M101B1Incomplete ,
	dutyStart:=M101B1Started ,
	standbyRemoteMode:=M101B2RemoteMode ,
	standbyOverload:=M101B2Overload ,
	standbyIncomplete:=M101B2Incomplete  ,
	standbyStart:=M101B2Started ,
	timeout:=T#2s ,
	dualMode:= TRUE,
	warningDutyOverload:=ADR(warning_M101B1Overload) ,
	warningDutyFailed:=ADR(warning_M101B1Failed) ,
	warningStandbyOverload:=ADR(warning_M101B2Overload) ,
	warningStandbyFailed:=ADR(warning_M101B2Failed) ,
	criticalErrorStartingFailed:=ADR(critical_M101BStartingFailed) ,
	criticalDutyStopFailed:= ADR(critical_M101B1StopFailed),
	criticalStandbyStopFailed:=ADR(critical_M101B2StopFailed),
	dutyCommand=>M101B1Command ,
	standbyCommand=>M101B2Command);





TANK_FOR_STREAM_1.LSD101A.IN;
TANK_FOR_STREAM_1.LSD101A.Q;
END_PROGRAM

(* POU module/blinker, FBD *)
FUNCTION_BLOCK blinker
VAR_INPUT
	IN: BOOL;
	OffTime: TIME := T#5m;
	OnTime: TIME:=T#2m;
END_VAR
VAR_OUTPUT
	Q: BOOL;
END_VAR
VAR
	tmr_off: TON;
	tmr_on: TON;
END_VAR
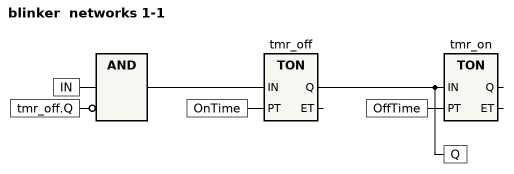
_FBD_ (* Function Block Diagram *)
NETWORK 1
	tmr_on:TON(IN: <tmr_off:TON(IN: AND(IN, NOT tmr_off.Q), PT: OnTime) => Q>, PT: OffTime)
_END_FBD_
END_FUNCTION_BLOCK

(* POU module/trigBlock, ST *)
FUNCTION_BLOCK trigBlock
VAR_INPUT
	IN:BOOL;
	aQ:POINTER TO BOOL;
END_VAR
VAR_OUTPUT
END_VAR
VAR
	inR_TRIG: R_TRIG;
	outF_TRIG: F_TRIG;
	Q: BOOL;
END_VAR
VAR_IN_OUT
END_VAR
IF aQ = 0 THEN
	aQ := ADR(Q);
END_IF


inR_TRIG(CLK:=IN );
outF_TRIG(CLK:=IN );

IF inR_TRIG.Q THEN
	aQ^ := TRUE;
ELSIF  outF_TRIG.Q THEN
	aQ^ := FALSE;
END_IF
END_FUNCTION_BLOCK
